// Mitsubishi GX Works2 project: fx3u-24MT   PLC: FX3U/FX3UC

PROGRAM MAIN
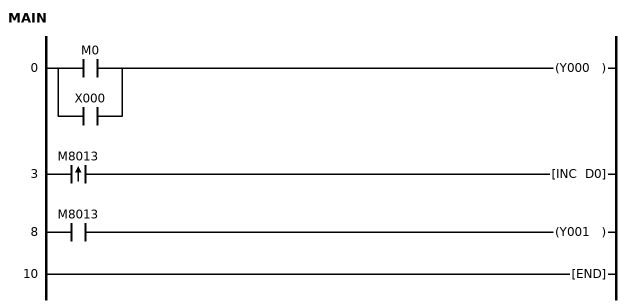
0     LD      M0
      OR      X000
      OUT     Y000
3     LDP     M8013
      INC     D0
8     LD      M8013
      OUT     Y001
10    END
END_PROGRAM
